// Mitsubishi GX Works2 project: test4   PLC: FX3U/FX3UC

PROGRAM MAIN
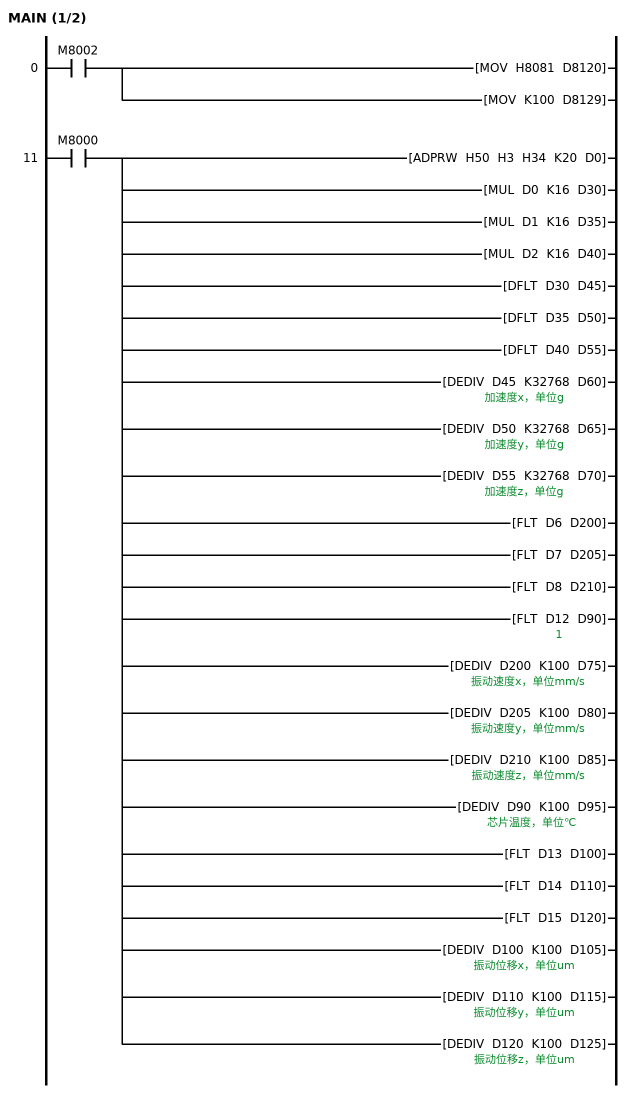
0     LD      M8002
      MOV     H8081 D8120
      MOV     K100 D8129
11    LD      M8000
      ADPRW   H50 H3 H34 K20 D0
      MUL     D0 K16 D30
      MUL     D1 K16 D35
      MUL     D2 K16 D40
      DFLT    D30 D45
      DFLT    D35 D50
      DFLT    D40 D55
      DEDIV   D45 K32768 D60  ; 加速度x，单位g
      DEDIV   D50 K32768 D65  ; 加速度y，单位g
      DEDIV   D55 K32768 D70  ; 加速度z，单位g
      FLT     D6 D200
      FLT     D7 D205
      FLT     D8 D210
      FLT     D12 D90  ; 1
      DEDIV   D200 K100 D75  ; 振动速度x，单位mm/s
      DEDIV   D205 K100 D80  ; 振动速度y，单位mm/s
      DEDIV   D210 K100 D85  ; 振动速度z，单位mm/s
      DEDIV   D90 K100 D95  ; 芯片温度，单位℃
      FLT     D13 D100
      FLT     D14 D110
      FLT     D15 D120
      DEDIV   D100 K100 D105  ; 振动位移x，单位um
      DEDIV   D110 K100 D115  ; 振动位移y，单位um
      DEDIV   D120 K100 D125  ; 振动位移z，单位um
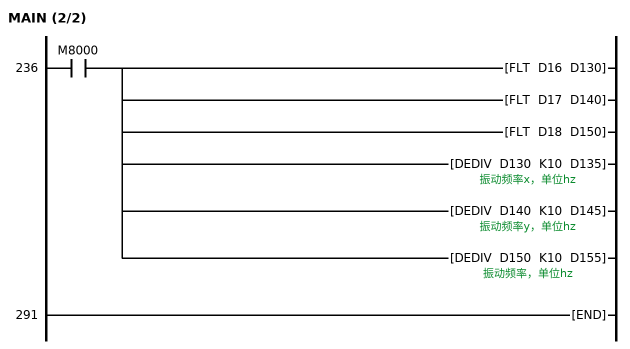
236   LD      M8000
      FLT     D16 D130
      FLT     D17 D140
      FLT     D18 D150
      DEDIV   D130 K10 D135  ; 振动频率x，单位hz
      DEDIV   D140 K10 D145  ; 振动频率y，单位hz
      DEDIV   D150 K10 D155  ; 振动频率，单位hz
291   END
END_PROGRAM

// device comments not shown above
D92  ; 转换浮点数温度
